{attribute 'enable_dynamic_creation'}
FUNCTION_BLOCK FB_EmptyObject IMPLEMENTS I_Object
VAR_INPUT
END_VAR
VAR_OUTPUT
END_VAR
VAR
	sObjectID			: STRING;
	eObjectType			: E_OBJECTS;
	// pointers for destructor
	_pInstance			: POINTER TO FB_EmptyObject;
	_pTemp				: POINTER TO FB_EmptyObject;
END_VAR

METHOD Destruct : BOOL
// destroy the instance 
IF _pInstance	<> 0 THEN
	// store in temp value otherwise the FB_exit called at __DELETE will create a stack overflow
	// when not set to 0 before __DELETE  
	_pTemp := _pInstance;
	_pInstance := 16#0; 
	__DELETE(_pTemp);
END_IF
END_METHOD

METHOD FB_exit : BOOL
VAR_INPUT
	bInCopyCode : BOOL; // if TRUE, the exit method is called for exiting an instance that is copied afterwards (online change).
END_VAR
Destruct();
END_METHOD

METHOD FB_init : BOOL
VAR_INPUT
	bInitRetains       : BOOL; // if TRUE, the retain variables are initialized (warm start / cold start)
	bInCopyCode        : BOOL;  // if TRUE, the instance afterwards gets moved into the copy code (online change)
	// Object identifier name
	sObjectID			: STRING;	
	// Object type as a string
	eObjectType			: E_OBJECTS;
END_VAR
THIS^.sObjectID		:= sObjectID;
THIS^.eObjectType	:= eObjectType;
END_METHOD

METHOD M_GetObjectDescription : string
VAR_INPUT
END_VAR
VAR
	sDescription			: STRING;
END_VAR
sDescription := concat(THIS^.sObjectID, ' Type: '); 
sDescription := concat(sDescription, TO_STRING(THIS^.eObjectType)); 
M_GetObjectDescription := sDescription;
END_METHOD

{warning 'add method implementation'}
METHOD M_Reset : BOOL
END_METHOD

{warning 'add method implementation'}
METHOD M_Start : BOOL
END_METHOD

{warning 'add property implementation'}
PROPERTY P_Status : DWORD
GET
END_GET
END_PROPERTY

PROPERTY pInstance : POINTER TO FB_EmptyObject
SET
// Store pointer for destructor
_pInstance := pInstance;
END_SET
END_PROPERTY

END_FUNCTION_BLOCK

(* stored: Version 1.1.0.1, ProductVersion 3.1.4024.12
   POU FB_EmptyObject: Id {233ae353-b7fc-445b-a060-dcc1d48d8608}, SpecialFunc None
   Method Destruct: Id {7662dfd7-e692-4980-be03-99e8c1af1a34}
   Method FB_exit: Id {46859754-a44e-4350-9673-1b2d304496b1}
   Method FB_init: Id {e9b051ea-6749-4848-88bc-65a2f326a012}
   Method M_GetObjectDescription: Id {9871546f-35e4-411d-9e77-65dd83e9ab96}
   Method M_Reset: Id {d0885b86-cac9-4d0a-98fe-ab2a0651959d}
   Method M_Start: Id {b40f8e59-0dae-42a4-918d-591c8f514f45}
   Property P_Status: Id {53684b99-8d1a-4b90-a247-c6e1693ac22f}
   Get Get: Id {d649fac2-415c-4875-a6da-507dff501e01}
   Property pInstance: Id {2f246fbe-2a73-4b22-bd6c-89ca2a9bc498}
   Set Set: Id {66b5e17f-da4c-470a-8eaa-c2460b2edcec} *)
